{attribute 'enable_dynamic_creation'}
FUNCTION_BLOCK FB_Black IMPLEMENTS I_Color
VAR_INPUT
END_VAR
VAR_OUTPUT
END_VAR
VAR
END_VAR


METHOD M_Fill : BOOL
ADSLOGSTR(ADSLOG_MSGTYPE_HINT, 'Paint Black', '');
M_Fill := TRUE;
END_METHOD

END_FUNCTION_BLOCK

(* stored: Version 1.1.0.1, ProductVersion 3.1.4024.12
   POU FB_Black: Id {25133850-c5b4-4409-ae57-f1dbf04be7a4}, SpecialFunc None
   Method M_Fill: Id {97774111-632e-441e-8ba9-2c360709bf52} *)
